(* IEC 61131-3 sources: volt/packages/volt-lsp-iec/test-corpus/bakon-nano/Device/Plc Logic/Application/Library Manager/(unresolved)/data server interfaces, 37 files *)

(* ---- DATASERVER_STRUCTREPLACEMENTINFO.dut ---- *)
TYPE DATASERVER_STRUCTREPLACEMENTINFO :
STRUCT
	PPARENTREPLACEMENTINFO : POINTER TO DataServer_StructReplacementInfo;
	ARRNAME : POINTER TO ARRAY [0..0] OF POINTER TO STRING(255);
	ARRREPLACEMENT : POINTER TO ARRAY [0..0] OF POINTER TO STRING(255);
	NCOUNT : INT;
END_STRUCT
END_TYPE

(* ---- DATASERVERFLAGS.dut ---- *)
TYPE DATASERVERFLAGS :
(
	NONE,
	FORINTEGRATEDVISU
);
END_TYPE

(* ---- DATASERVERREQUESTIDENTIFICATION.dut ---- *)
TYPE DATASERVERREQUESTIDENTIFICATION :
(
	NONE,
	ALARMSGETCOUNT,
	ALARMSGETALARMS
);
END_TYPE

(* ---- DATASOURCESHUTDOWNFLAGS.dut ---- *)
TYPE DATASOURCESHUTDOWNFLAGS :
(
	SUCCEEDED := 16#0,
	TIMEOUTOCCURRED := 16#1
);
END_TYPE

(* ---- DATASOURCESTATE.dut ---- *)
TYPE DATASOURCESTATE :
(
	DS_NEW,
	DS_INITIALIZED,
	DS_CONNECTING,
	DS_READY,
	DS_BUSY,
	DS_SHUTTINGDOWN,
	DS_SHUTDOWN,
	DS_ERROR
);
END_TYPE

(* ---- DATASOURCETRANSACTIONRESULT.dut ---- *)
TYPE DATASOURCETRANSACTIONRESULT :
(
	TR_OK,
	TR_PENDING,
	TR_UNKNOWNTRANSACTION,
	TR_ERROR
);
END_TYPE

(* ---- DRIVERINITINFO.dut ---- *)
TYPE DRIVERINITINFO :
STRUCT
	DWDATATAG : DWORD;
	DWDATAVERSION : DWORD;
	DWDATASIZE : DWORD;
END_STRUCT
END_TYPE

(* ---- PLCADDRESSINFOUNION.dut ---- *)
TYPE PLCADDRESSINFOUNION :
UNION
	COMMON : PlcAddressInfo;
	ABSOLUTE : PlcAbsoluteAddressInfo;
	PROPBYCALL : PlcPropertyByCallAddressInfo;
END_UNION
END_TYPE

(* ---- SWAPPINGINFO.dut ---- *)
TYPE SWAPPINGINFO :
(
	NOSWAPPINGNEEDED := 0,
	SWAPPINGNEEDED := 1,
	UNKNOWN := -1,
	APPLICATIONNOTFOUND := -2,
	INTERFACENOTIMPLEMENTED := -3
);
END_TYPE

(* ---- TYPEIDS.dut ---- *)
TYPE TYPEIDS :
(
	DATASERVERDATAITEMLIST := 1,
	DATASERVERACTIONRECORD := 2
);
END_TYPE

(* ---- DATAITEMQUALITYCODES.gvl ---- *)
VAR_GLOBAL
	MASK_LOWESTLEVEL : DWORD := 16#FFFF;
	MASK_DRIVERLEVEL : DWORD := 16#FF0000;
	MASK_APPLICATIONLEVEL : DWORD := 16#FF000000;
	APPLEVEL_LASTUPDATEFAILED : DWORD := 16#1000000;
	APPLEVEL_TIMEOUT : DWORD := 16#2000000;
END_VAR

(* ---- DATASERVERSETTINGS.gvl ---- *)
VAR_GLOBAL
	TAG_TIMEOUT_DRIVERBUSY : DWORD := 16#1;
	TAG_TIMEOUT_DRIVERSYNCSHUTDOWN : DWORD := 16#2;
	TAG_TIMESLICE_DRIVERSYNCSHUTDOWN : DWORD := 16#3;
	TAG_RECOVER_RECONNECTWAITTIME : DWORD := 16#4;
	TAG_RECOVER_ERRORWAITTIME : DWORD := 16#5;
	TAG_RECOVER_RECONNECTBUSYTIMEOUTWAITTIME : DWORD := 16#6;
	TAG_RECOVER_IDENTITYMISMATCH : DWORD := 16#7;
	TAG_MEMORY_STARTRESERVEREADITEMS : DWORD := 16#8;
	TAG_MEMORY_STARTRESERVEWRITEITEMS : DWORD := 16#9;
	TAG_RECOVER_RECONNECTCURRENTWAITTIME : DWORD := 16#A;
	TAG_UPDATEINSTOPMODE : DWORD := 16#B;
	DEFAULT_TIMEOUT_DRIVERBUSY : DWORD := 5000;
	DEFAULT_TIMEOUT_DRIVERSYNCSHUTDOWN : DWORD := 3000;
	DEFAULT_TIMESLICE_DRIVERSYNCSHUTDOWN : DWORD := 100;
	DEFAULT_RECOVER_RECONNECTWAITTIME : DWORD := 20000;
	DEFAULT_RECOVER_ERRORWAITTIME : DWORD := 30000;
	DEFAULT_RECOVER_RECONNECTBUSYTIMEOUTWAITTIME : DWORD := 3000;
	DEFAULT_RECOVER_IDENTITYMISMATCH : DWORD := 120000;
	DEFAULT_RECOVER_RECONNECTCURRENTWAITTIME : DWORD := 0;
	DEFAULT_UPDATEINSTOPMODE : DWORD := 0;
	DEFAULT_MEMORY_STARTRESERVEREADITEMS : DWORD := 100;
	DEFAULT_MEMORY_STARTRESERVEWRITEITEMS : DWORD := 100;
END_VAR

(* ---- DRIVERINITCONSTANTS.gvl ---- *)
VAR_GLOBAL
	CUSTOMERMASK : DWORD := 16#FFFF0000;
	DRIVERMASK : DWORD := 16#FFFF;
	CUSTOMER_STANDARD : WORD := 16#0;
	DRIVER_UNKNOWN : WORD := 16#0;
	DRIVER_MONITORING_STANDARD : WORD := 16#1;
	DRIVER_OPC_STANDARD : WORD := 16#2;
	DRIVER_SYMBOLICMONITORING_STANDARD : WORD := 16#3;
END_VAR

(* ---- INTERFACEIDS.gvl ---- *)
VAR_GLOBAL
	ITFID_IGENERIC : DWORD := 0;
	ITFID_IDATASERVER : DWORD := 1;
	ITFID_IDATASERVER2 : DWORD := 2;
	ITFID_ICREDENTIALSPROVIDER : DWORD := 3;
	ITFID_IDATASOURCEDRIVER : DWORD := 4;
	ITFID_IDATASOURCEDRIVER2 : DWORD := 5;
	ITFID_IDATASOURCEDRIVER3 : DWORD := 6;
	ITFID_IDATASERVER3 : DWORD := 7;
	ITFID_IDATASERVER4 : DWORD := 8;
	ITFID_ICALLBACK : DWORD := 9;
	ITFID_IDATAITEMLIST : DWORD := 10;
	ITFID_IPROVIDESCONCRETETYPE : DWORD := 11;
	ITFID_IDATASOURCEDRIVER4 : DWORD := 12;
	ITFID_IDATASERVER5 : DWORD := 13;
	ITFID_ITEMPSHUTDOWNRESULT : DWORD := 14;
	ITFID_IDATASERVERACTIONRECORD : DWORD := 15;
	ITFID_IDATASOURCEDRIVER5 : DWORD := 16;
	ITFID_IDATASERVER6 : DWORD := 17;
END_VAR

(* ---- RETURNVALUES.gvl ---- *)
VAR_GLOBAL
	ERR_OK : UDINT := 16#0;
	ERR_FAILED : UDINT := 16#1;
	ERR_PARAMETER : UDINT := 16#2;
	ERR_NOTINITIALIZED : UDINT := 16#3;
	ERR_VERSION : UDINT := 16#4;
	ERR_TIMEOUT : UDINT := 16#5;
	ERR_NOBUFFER : UDINT := 16#6;
	ERR_PENDING : UDINT := 16#A;
	ERR_NUMPENDING : UDINT := 16#B;
	ERR_NOTIMPLEMENTED : UDINT := 16#C;
	ERR_INVALIDID : UDINT := 16#D;
	ERR_OVERFLOW : UDINT := 16#E;
	ERR_BUFFERSIZE : UDINT := 16#F;
	ERR_NO_OBJECT : UDINT := 16#10;
	ERR_NOMEMORY : UDINT := 16#11;
	ERR_DUPLICATE : UDINT := 16#12;
	ERR_INVALID_HANDLE : UDINT := 16#14;
	ERR_NO_CHANGE : UDINT := 16#16;
	ERR_INVALID_INTERFACE : UDINT := 16#17;
	ERR_NOT_SUPPORTED : UDINT := 16#18;
	ERR_OUT_OF_LIMITS : UDINT := 16#1A;
	ERR_DS_UNKNOWN : UDINT := 16#2000;
	ERR_DS_UNKNOWN_GROUP : UDINT := 16#2001;
	ERR_DS_UNKNOWN_SYMBOL : UDINT := 16#2002;
	ERR_DS_UNKNOWN_TRANSACTION : UDINT := 16#2003;
	ERR_DS_INVALID_STATE : UDINT := 16#2004;
	ERR_DS_INVALID_PATH : UDINT := 16#2005;
	ERR_DS_SOURCENOTFOUND : UDINT := 16#2006;
	ERR_DS_ITEMNOTFOUND : UDINT := 16#2007;
	ERR_DS_MULTITASKING_LOCKED : UDINT := 16#2008;
	ERR_DS_TIMEOUT : UDINT := 16#2009;
	ERR_DS_BADITEMS : UDINT := 16#200A;
	ERR_DS_ITEMNOTACTIVE : UDINT := 16#200B;
	ERR_DS_RETRYLOGIN : UDINT := 16#200C;
	ERR_DSD_IDENTITY_MISMATCH : UDINT := 16#2100;
	ERR_DSD_LOGINFAILED : UDINT := 16#2101;
	ERR_DSD_LOGINNECESSARY : UDINT := 16#2102;
END_VAR

(* ---- ICALLBACK.itf ---- *)
INTERFACE ICALLBACK
END_INTERFACE

METHOD CALLBACK
VAR_INPUT
	PPARAM : POINTER TO BYTE;
END_VAR
END_METHOD

(* ---- ICREDENTIALSPROVIDER.itf ---- *)
INTERFACE ICREDENTIALSPROVIDER
END_INTERFACE

METHOD GETCREDENTIALS : UDINT
VAR_INPUT
	UDIREQUESTID : UDINT;
END_VAR
VAR_OUTPUT
	STUSERNAME : STRING;
	STPASSWORD : STRING;
END_VAR
END_METHOD

METHOD ISGETCREDENTIALSFINISHED : UDINT
VAR_INPUT
	UDIREQUESTID : UDINT;
END_VAR
END_METHOD

METHOD LOGINFAILED : UDINT
VAR_INPUT
	UDIREQUESTID : UDINT;
END_VAR
VAR_OUTPUT
	UDIRETRYWAITTIME : UDINT;
END_VAR
END_METHOD

METHOD STARTGETCREDENTIALS : UDINT
VAR_INPUT
	PSTDATASOURCE : POINTER TO STRING;
END_VAR
VAR_OUTPUT
	UDIERRORCODE : UDINT;
END_VAR
END_METHOD

(* ---- IDATAGROUP.itf ---- *)
INTERFACE IDATAGROUP
END_INTERFACE

METHOD ADDITEM : UDINT
VAR_INPUT
	PSTSYMBOL : POINTER TO STRING;
END_VAR
END_METHOD

METHOD CLEAR : BOOL
END_METHOD

METHOD RELEASE : UDINT
END_METHOD

METHOD USE : UDINT
END_METHOD

(* ---- IDATAITEMLIST.itf ---- *)
INTERFACE IDATAITEMLIST
END_INTERFACE

METHOD CLEAR : UDINT
END_METHOD

METHOD CREATEANDADD : UDINT
VAR_INPUT
	PSTINSTANCEPATH : POINTER TO BYTE;
END_VAR
VAR_OUTPUT
	CREATEDITEM : IDataItem2;
END_VAR
END_METHOD

METHOD GETITEM : IDataItem2
VAR_INPUT
	UDIINDEX : UDINT;
END_VAR
END_METHOD

(* ---- IDATASERVER.itf ---- *)
INTERFACE IDATASERVER
END_INTERFACE

METHOD ALLITEMSOK : UDINT
END_METHOD

METHOD BEGINDATACONFIGURATION : UDINT
VAR_INPUT
	BBLOCKING : BOOL;
END_VAR
END_METHOD

METHOD ENDDATACONFIGURATION : UDINT
END_METHOD

METHOD GETITEMINFO : IDataItemInfo
VAR_INPUT
	PSTSYMBOL : POINTER TO STRING;
END_VAR
VAR_OUTPUT
	UDIRESULT : UDINT;
END_VAR
END_METHOD

METHOD RELEASEDATA : UDINT
VAR_INPUT
	PSTSYMBOL : POINTER TO STRING;
END_VAR
END_METHOD

METHOD USEDATA : UDINT
VAR_INPUT
	PSTSYMBOL : POINTER TO STRING;
END_VAR
END_METHOD

(* ---- IDATASERVER2.itf ---- *)
INTERFACE IDATASERVER2
END_INTERFACE

METHOD GETINTERFACE : POINTER TO BYTE
VAR_INPUT
	DWITFID : DWORD;
END_VAR
END_METHOD

METHOD SETCREDENTIALSPROVIDER : UDINT
VAR_INPUT
	PSTDATASOURCE : POINTER TO STRING;
	CREDPROV : ICredentialsProvider;
END_VAR
END_METHOD

(* ---- IDATASERVER3.itf ---- *)
INTERFACE IDATASERVER3
END_INTERFACE

METHOD RESOLVESYMBOL : UDINT
VAR_INPUT
	PSTSYMBOL : POINTER TO BYTE;
END_VAR
VAR_OUTPUT
	PLOCAL : POINTER TO BYTE;
	ITEMTYPE : PlcDataItemType;
	PADDRINFO : POINTER TO PlcAddressInfo;
END_VAR
END_METHOD

(* ---- IDATASERVER4.itf ---- *)
INTERFACE IDATASERVER4
END_INTERFACE

METHOD CREATEITEMLIST : IDataItemList
VAR_INPUT
	UDIINITIALCAPACITY : UDINT;
END_VAR
END_METHOD

METHOD DELETEITEMLIST : UDINT
VAR_INPUT
	ITEMSLIST : IDataItemList;
END_VAR
END_METHOD

METHOD READITEMS : UDINT
VAR_INPUT
	ITEMS : IDataItemList;
	BASYNCHRON : BOOL;
	FINISHEDCALLBACK : ICallback;
END_VAR
END_METHOD

METHOD WRITEITEMS : UDINT
VAR_INPUT
	ITEMS : IDataItemList;
	BASYNCHRON : BOOL;
	FINISHEDCALLBACK : ICallback;
END_VAR
END_METHOD

(* ---- IDATASERVER5.itf ---- *)
INTERFACE IDATASERVER5
END_INTERFACE

METHOD DELETERECORD : UDINT
VAR_INPUT
	RECORD : IDataServerActionRecord;
END_VAR
END_METHOD

METHOD GETRECORDRESULT : UDINT
VAR_OUTPUT
	RESULT : IDataServerActionRecord;
END_VAR
END_METHOD

METHOD REPLAYRECORD : UDINT
VAR_INPUT
	RECORD : IDataServerActionRecord;
END_VAR
END_METHOD

METHOD RESUMEAFTERTEMPSHUTDOWN : UDINT
VAR_INPUT
	PSTDATASOURCE : POINTER TO STRING;
END_VAR
END_METHOD

METHOD STARTRECORDMODE : UDINT
END_METHOD

METHOD STARTTEMPSHUTDOWN : UDINT
VAR_INPUT
	PSTDATASOURCE : POINTER TO STRING;
	CBSHUTDOWNDONE : ICallback;
END_VAR
END_METHOD

(* ---- IDATASERVER6.itf ---- *)
INTERFACE IDATASERVER6
END_INTERFACE

METHOD GETADDRESS : UDINT
VAR_INPUT
	PSTSYMBOL : POINTER TO STRING;
END_VAR
VAR_OUTPUT
	ADDRESS : PlcAddressInfoUnion;
END_VAR
END_METHOD

METHOD ISSWAPPINGNEEDED : SwappingInfo
VAR_INPUT
	SNAME : STRING;
END_VAR
END_METHOD

METHOD PROCESSDATASERVERREQUEST : UDINT
VAR_INPUT
	SNAME : STRING;
	ITFREQUESTPARAMETER : IRequestParameter;
	ITFREQUESTRESULT : IRequestResult;
	DIREQUESTID : DINT;
END_VAR
END_METHOD

(* ---- IDATASERVERACTIONRECORD.itf ---- *)
INTERFACE IDATASERVERACTIONRECORD
END_INTERFACE

(* ---- IDATASERVERFRAMEMANAGER.itf ---- *)
INTERFACE IDATASERVERFRAMEMANAGER
END_INTERFACE

METHOD GETCOUNT : INT
END_METHOD

METHOD GETREPLACEDPATH : POINTER TO STRING(255)
VAR_INPUT
	PSTINTERFACEVAR : POINTER TO STRING(255);
	PREPLACEMENTINFO : POINTER TO DataServer_StructReplacementInfo;
END_VAR
END_METHOD

METHOD GETREPLACEMENTINFO : POINTER TO DataServer_StructReplacementInfo
VAR_INPUT
	PSTFRAMEPATH : POINTER TO STRING(255);
END_VAR
END_METHOD

(* ---- IDATASOURCEDRIVER.itf ---- *)
INTERFACE IDATASOURCEDRIVER
END_INTERFACE

METHOD CONNECTING : UDINT
END_METHOD

METHOD GETREQUESTRESULT : DataSourceTransactionResult
VAR_INPUT
	DWTRANSACTIONID : DWORD;
END_VAR
END_METHOD

METHOD GETSETTING : DWORD
VAR_INPUT
	DWSETTINGTAG : DWORD;
END_VAR
VAR_OUTPUT
	BUSEDEFAULT : BOOL;
END_VAR
END_METHOD

METHOD INITIALIZE : UDINT
VAR_INPUT
	STDATASOURCE : STRING;
	PINITINFO : POINTER TO DriverInitInfo;
	PINITDATA : POINTER TO BYTE;
END_VAR
END_METHOD

METHOD READREQUEST : UDINT
VAR_INPUT
	PITEMS : POINTER TO ARRAY [0..100] OF IDataItem;
	IITEMCOUNT : UDINT;
	DWLISTID : DWORD;
END_VAR
VAR_OUTPUT
	DWTRANSACTIONID : DWORD;
END_VAR
END_METHOD

METHOD RESET : UDINT
END_METHOD

METHOD SHUTTINGDOWN : UDINT
END_METHOD

METHOD STARTCONNECT : UDINT
END_METHOD

METHOD STARTSHUTDOWN : UDINT
END_METHOD

METHOD UPDATEREQUEST : UDINT
VAR_INPUT
	PITEMS : POINTER TO ARRAY [0..100] OF IDataItem;
	IITEMCOUNT : UDINT;
	DWLISTID : DWORD;
	DWTRANSACTIONID : DWORD;
END_VAR
END_METHOD

METHOD WRITEREQUEST : UDINT
VAR_INPUT
	PITEMS : POINTER TO ARRAY [0..100] OF IDataItem;
	IITEMCOUNT : UDINT;
	DWLISTID : DWORD;
END_VAR
VAR_OUTPUT
	DWTRANSACTIONID : DWORD;
END_VAR
END_METHOD

(* ---- IDATASOURCEDRIVER2.itf ---- *)
INTERFACE IDATASOURCEDRIVER2
END_INTERFACE

METHOD SHUTDOWNFINISHED : UDINT
VAR_INPUT
	DWFLAGS : DWORD;
END_VAR
END_METHOD

(* ---- IDATASOURCEDRIVER3.itf ---- *)
INTERFACE IDATASOURCEDRIVER3
END_INTERFACE

METHOD ASSIGNCREDENTIALS : UDINT
VAR_INPUT
	STUSERNAME : STRING;
	STPASSWORD : STRING;
END_VAR
END_METHOD

METHOD GETINTERFACE : POINTER TO BYTE
VAR_INPUT
	DWITFID : DWORD;
END_VAR
END_METHOD

(* ---- IDATASOURCEDRIVER4.itf ---- *)
INTERFACE IDATASOURCEDRIVER4
END_INTERFACE

METHOD READREQUEST2 : UDINT
VAR_INPUT
	PITEMS : POINTER TO ARRAY [0..100] OF IDataItem;
	IITEMCOUNTTOTAL : UDINT;
	ISTARTOFFSET : UDINT;
	DWLISTID : DWORD;
END_VAR
VAR_OUTPUT
	DWTRANSACTIONID : DWORD;
	ISENTITEMS : UDINT;
END_VAR
END_METHOD

METHOD WRITEREQUEST2 : UDINT
VAR_INPUT
	PITEMS : POINTER TO ARRAY [0..100] OF IDataItem;
	IITEMCOUNTTOTAL : UDINT;
	ISTARTOFFSET : UDINT;
	DWLISTID : DWORD;
END_VAR
VAR_OUTPUT
	DWTRANSACTIONID : DWORD;
	ISENTITEMS : UDINT;
END_VAR
END_METHOD

(* ---- IDATASOURCEDRIVER5.itf ---- *)
INTERFACE IDATASOURCEDRIVER5
END_INTERFACE

METHOD ISSWAPPINGNEEDED : SwappingInfo
END_METHOD

METHOD PROCESSDATASERVERREPLY : UDINT
VAR_INPUT
	DWTRANSACTIONID : DWORD;
	ITFREQUESTPARAMETER : IRequestParameter;
	ITFREQUESTRESULT : IRequestResult;
END_VAR
END_METHOD

METHOD PROCESSDATASERVERREQUEST : UDINT
VAR_INPUT
	ITFREQUESTPARAMETER : IRequestParameter;
END_VAR
VAR_OUTPUT
	DWTRANSACTIONID : DWORD;
END_VAR
END_METHOD

(* ---- IGENERIC.itf ---- *)
INTERFACE IGENERIC
END_INTERFACE

METHOD GETINTERFACE : POINTER TO BYTE
VAR_INPUT
	DWITFID : DWORD;
END_VAR
END_METHOD

(* ---- IPROVIDESCONCRETETYPE.itf ---- *)
INTERFACE IPROVIDESCONCRETETYPE
END_INTERFACE

(* ---- IREQUESTPARAMETER.itf ---- *)
INTERFACE IREQUESTPARAMETER
END_INTERFACE

METHOD GETREQUESTIDENTIFICATION : DataServerRequestIdentification
END_METHOD

(* ---- IREQUESTRESULT.itf ---- *)
INTERFACE IREQUESTRESULT
END_INTERFACE

METHOD ISREPLYPENDING : BOOL
END_METHOD

METHOD SETREPLYPENDING
VAR_INPUT
	XREPLYPENDING : BOOL;
END_VAR
END_METHOD

(* ---- ITEMPSHUTDOWNRESULT.itf ---- *)
INTERFACE ITEMPSHUTDOWNRESULT
END_INTERFACE
